PROGRAM BkgrdSerialOpticalPowermeterHs
VAR
	(* background communication with the EL6002 terminal *)
	serialLineCtrl		: SerialLineControl;
	serialLineCtrlError	: BOOL;
	serialLineCtrlErrorID : ComError_t;
	(* 	I/O variables for a EL6002 terminal*)
	stInThorlabsOpticalPowermeterHs  AT %I* : EL6inData22B;	
	stOutThorlabsOpticalPowermeterHs AT %Q* : EL6outData22B;
END_VAR

(*
The SerialLineControl function block is supposed to be called in every PLC cycle.
It communicates with the serial line hardware device and transmits or receives data.
The SerialLineControl can be called in the standard task (e.g.for PcCOM port usage) 
or in a separate fast task (e.g.for terminal usage) as well.
A fast separate task will be necessary at high baud rates or with KL6001 terminals 
which have a small process image (3 or 5 data bytes only)
*)

(* background communication with the EL6002 terminal *)
serialLineCtrl(
	Mode:= SERIALLINEMODE_EL6_22B, 
	pComIn:= ADR(stInThorlabsOpticalPowermeterHs), 
	pComOut:= ADR(stOutThorlabsOpticalPowermeterHs), 
	SizeComIn:= SIZEOF(stInThorlabsOpticalPowermeterHs), 
	TxBuffer:= HardwareGlobalVariables.TxBufferOpticalPowermeterHs, 
	RxBuffer:= HardwareGlobalVariables.RxBufferOpticalPowermeterHs
);

IF serialLineCtrl.Error THEN
	serialLineCtrlError := TRUE;
	serialLineCtrlErrorID := serialLineCtrl.ErrorID;
END_IF

END_PROGRAM

(* stored: Version 1.1.0.1, ProductVersion 3.1.4024.4
   POU BkgrdSerialOpticalPowermeterHs: Id {06a32bf0-813e-4602-8c55-1c491d4f8144}, SpecialFunc None *)
